// TIA Portal V18 export
ORGANIZATION_BLOCK "PID Control Valve"   // OB30, LAD, CyclicInterrupt
{ S7_Optimized_Access := 'TRUE' }
VERSION : 0.1
// stored: AutoNumber true, IsIECCheckEnabled false, SetENOAutomatically false
   VAR_INPUT
      Initial_Call : Bool;   // Initial call of this OB
      Event_Count : Int;   // Events discarded
   END_VAR
BEGIN

REGION Network 1: Put the variables for the pid
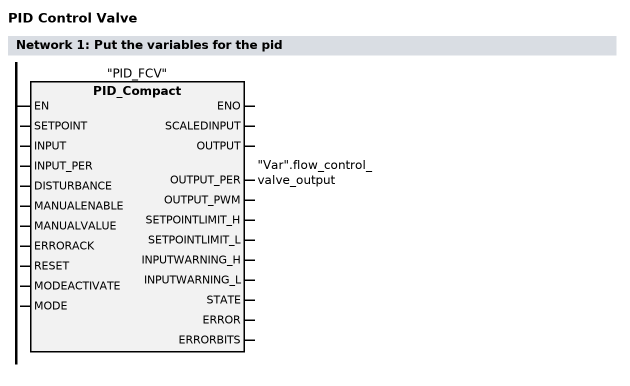
   RUNG wire#powerrail
      "PID_FCV".PID_Compact(Setpoint :=, Input :=, Input_PER :=, Disturbance :=, ManualEnable :=, ManualValue :=, ErrorAck :=, Reset :=, ModeActivate :=, Mode :=, ScaledInput =>, Output =>, Output_PER => "Var".flow_control_valve_output, Output_PWM =>, SetpointLimit_H =>, SetpointLimit_L =>, InputWarning_H =>, InputWarning_L =>, State =>, Error =>, ErrorBits =>)
   END_RUNG
   // the same network as SCL:
   "PID_FCV"(Output_PER => "Var".flow_control_valve_output);   // PID_Compact
END_REGION
END_ORGANIZATION_BLOCK
